// Mitsubishi GX Works2 project: 20240117_AI机程序新增旋钮开关-BACKUP   PLC: FX3S

PROGRAM MAIN
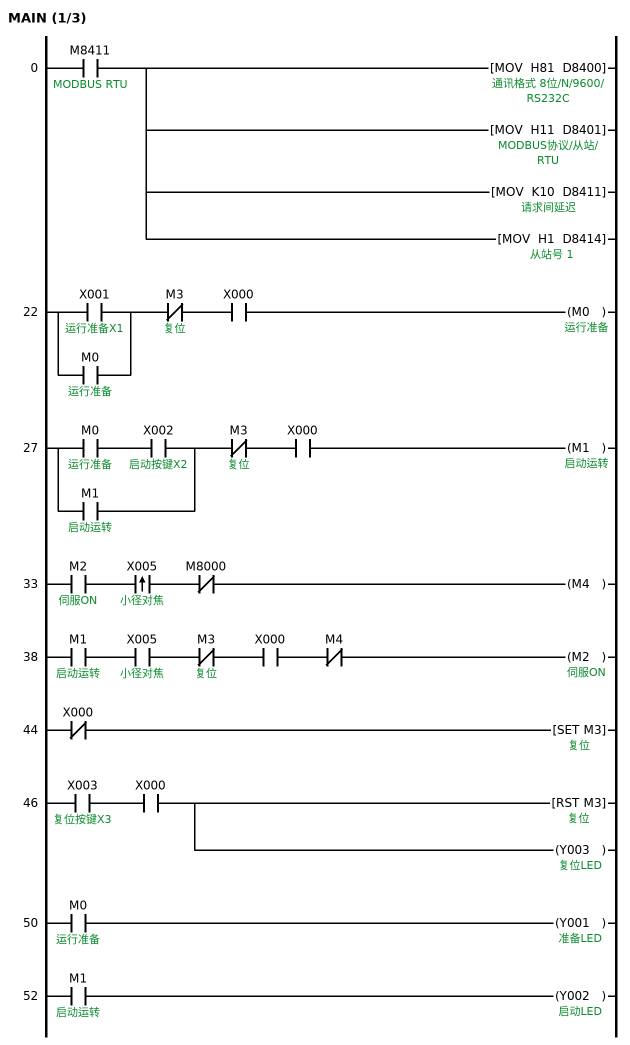
0     LD      M8411  ; MODBUS RTU
      MOV     H81 D8400  ; 通讯格式 8位/N/9600/RS232C
      MOV     H11 D8401  ; MODBUS协议/从站/RTU
      MOV     K10 D8411  ; 请求间延迟
      MOV     H1 D8414  ; 从站号 1
22    LD      X001  ; 运行准备X1
      OR      M0  ; 运行准备
      ANI     M3  ; 复位
      AND     X000
      OUT     M0  ; 运行准备
27    LD      M0  ; 运行准备
      AND     X002  ; 启动按键X2
      OR      M1  ; 启动运转
      ANI     M3  ; 复位
      AND     X000
      OUT     M1  ; 启动运转
33    LD      M2  ; 伺服ON
      ANDP    X005  ; 小径对焦
      ANI     M8000
      OUT     M4
38    LD      M1  ; 启动运转
      AND     X005  ; 小径对焦
      ANI     M3  ; 复位
      AND     X000
      ANI     M4
      OUT     M2  ; 伺服ON
44    LDI     X000
      SET     M3  ; 复位
46    LD      X003  ; 复位按键X3
      AND     X000
      RST     M3  ; 复位
      OUT     Y003  ; 复位LED
50    LD      M0  ; 运行准备
      OUT     Y001  ; 准备LED
52    LD      M1  ; 启动运转
      OUT     Y002  ; 启动LED
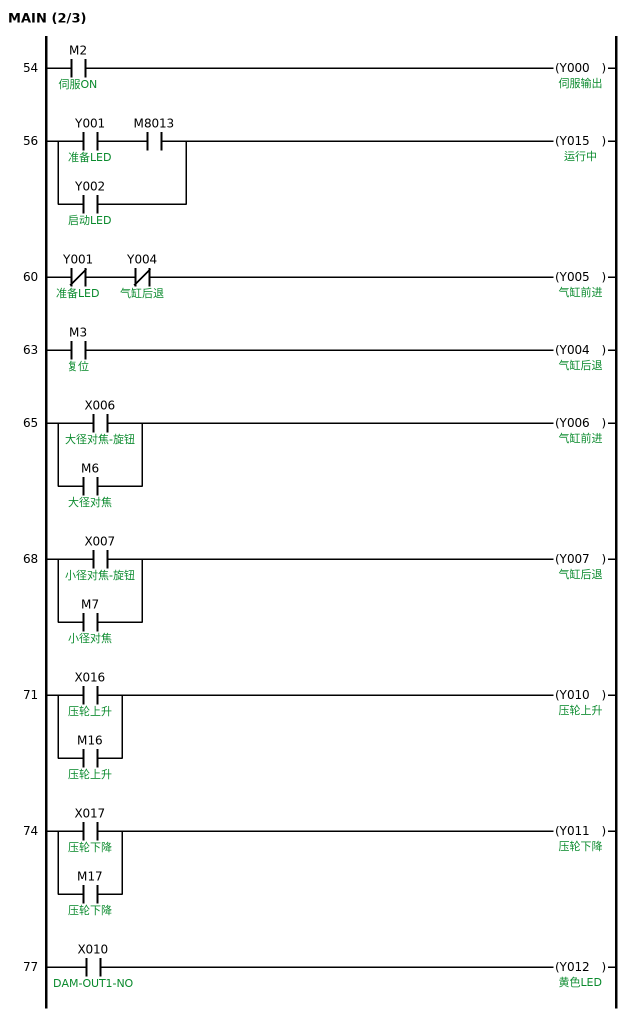
54    LD      M2  ; 伺服ON
      OUT     Y000  ; 伺服输出
56    LD      Y001  ; 准备LED
      AND     M8013
      OR      Y002  ; 启动LED
      OUT     Y015  ; 运行中
60    LDI     Y001  ; 准备LED
      ANI     Y004  ; 气缸后退
      OUT     Y005  ; 气缸前进
63    LD      M3  ; 复位
      OUT     Y004  ; 气缸后退
65    LD      X006  ; 大径对焦-旋钮
      OR      M6  ; 大径对焦
      OUT     Y006  ; 气缸前进
68    LD      X007  ; 小径对焦-旋钮
      OR      M7  ; 小径对焦
      OUT     Y007  ; 气缸后退
71    LD      X016  ; 压轮上升
      OR      M16  ; 压轮上升
      OUT     Y010  ; 压轮上升
74    LD      X017  ; 压轮下降
      OR      M17  ; 压轮下降
      OUT     Y011  ; 压轮下降
77    LD      X010  ; DAM-OUT1-NO
      OUT     Y012  ; 黄色LED
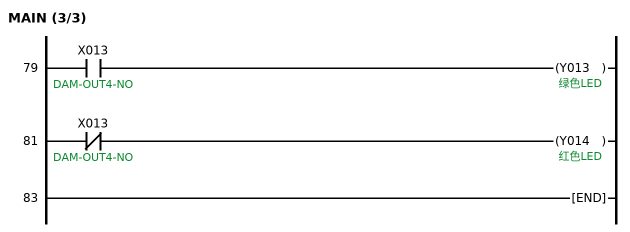
79    LD      X013  ; DAM-OUT4-NO
      OUT     Y013  ; 绿色LED
81    LDI     X013  ; DAM-OUT4-NO
      OUT     Y014  ; 红色LED
83    END
END_PROGRAM

// device comments not shown above
X011  ; DAM-OUT2-NO
X012  ; DAM-OUT3-NO
X014  ; DAM-OUT5-NO
X015  ; DAM-OUT6-NO
